// TIA Portal V18 export
FUNCTION "mot_speed_by_target" : Void   // FC7, FBD
{ S7_Optimized_Access := 'TRUE' }
VERSION : 0.1
// stored: AutoNumber true, IsIECCheckEnabled false, SetENOAutomatically false, UDAEnableTagReadback false
   VAR_INPUT
      isMultiturn : Bool;
      MultiTurnGoesFwdOnly : Bool;
      SET_SPD_ABS : Real;
      POS : Real;
      TARGET : Real;
      par_lim_fwd : Real;
      par_lim_rev : Real;
      par_speed_absmax : Real;
      par_dist_absmax : Real;
      par_speed_crawl : Real;
      par_dist_crawl : Real;
      par_dist_stop : Real;
   END_VAR
   VAR_OUTPUT
      speed_dir : Real;
      ER : Bool;
      ER_W : WString;
   END_VAR
   VAR_TEMP
      target_plus_TURN : Real;
      target_minus_TURN : Real;
      target_local : Real;
      dir_fwd : Bool;
      dir_rev : Bool;
      speed_fwd : Real;
      speed_rev : Real;
      set_spd_w_dir : Real;
      turn : Real;
      dist_to_target : Real;
      dist_to_target_plus_turn : Real;
      dist_to_target_minus_turn : Real;
      distance1 : Real;
      distance2plus : Real;
      turn_inv : Real;
      distance3minus : Real;
      closest0 : Bool;
      closest1Plus : Bool;
      closest2Minus : Bool;
      target_normal : Real;
   END_VAR
BEGIN

REGION Network 2 (SCL)
   IF "ER_0_root".ACK THEN
       #ER_W := WSTRING#'';
       #ER := false;

   END_IF;
   #turn := #par_lim_fwd - #par_lim_rev;
   #turn_inv := - #turn;
END_REGION

REGION Network 3
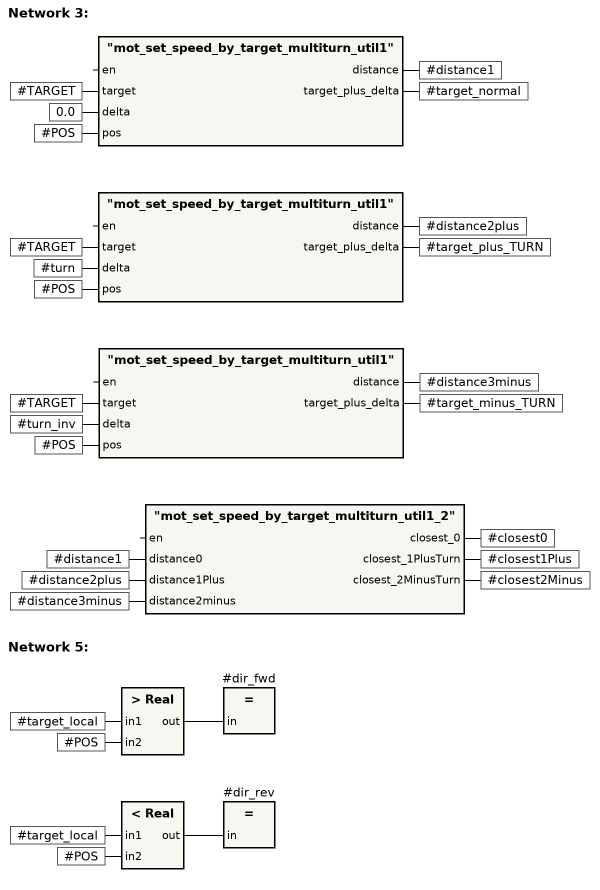
   "mot_set_speed_by_target_multiturn_util1"(target := #TARGET,
                           delta := 0.0,
                           pos := #POS,
                           distance => #distance1,
                           target_plus_delta => #target_normal);
   "mot_set_speed_by_target_multiturn_util1"(target := #TARGET,
                           delta := #turn,
                           pos := #POS,
                           distance => #distance2plus,
                           target_plus_delta => #target_plus_TURN);
   "mot_set_speed_by_target_multiturn_util1"(target := #TARGET,
                           delta := #turn_inv,
                           pos := #POS,
                           distance => #distance3minus,
                           target_plus_delta => #target_minus_TURN);
   "mot_set_speed_by_target_multiturn_util1_2"(distance0 := #distance1,
                           distance1Plus := #distance2plus,
                           distance2minus := #distance3minus,
                           closest_0 => #closest0,
                           closest_1PlusTurn => #closest1Plus,
                           closest_2MinusTurn => #closest2Minus);
END_REGION

REGION Network 4 (SCL)
   IF #isMultiturn AND NOT #ER THEN
       IF #MultiTurnGoesFwdOnly THEN
           IF #closest1Plus THEN
               #target_local := #target_plus_TURN;
           ELSE
               #target_local := #target_normal;
           END_IF;
       ELSE
           IF #closest1Plus THEN
               #target_local := #target_plus_TURN;
           ELSIF #closest2Minus THEN
               #target_local := #target_minus_TURN;
           ELSE
               #target_local := #target_normal;
           END_IF;
       END_IF;


   ELSE
       #target_local := #TARGET;
   END_IF;
END_REGION

REGION Network 5
   #dir_fwd := #target_local > #POS;
   #dir_rev := #target_local < #POS;
END_REGION

REGION Network 6
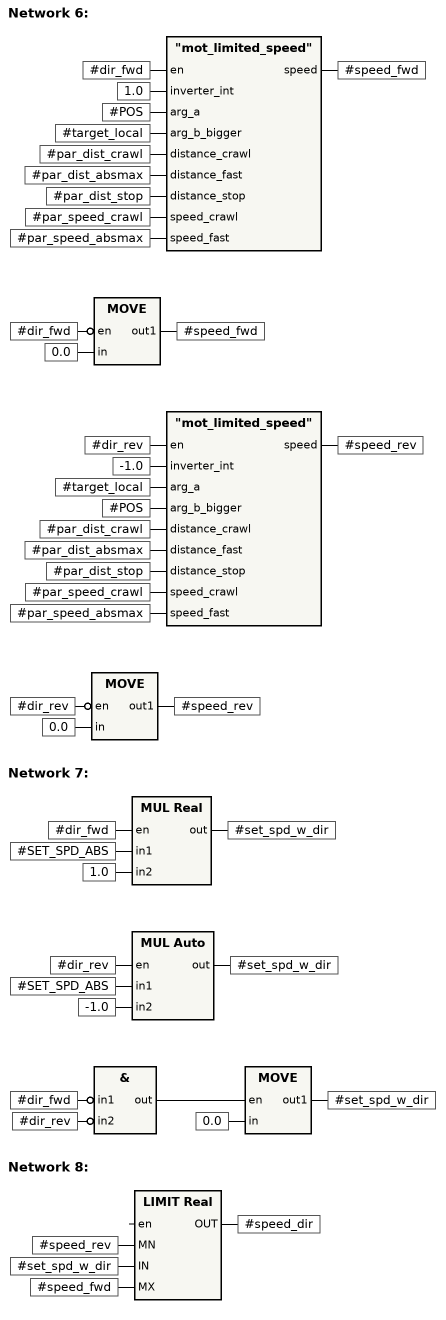
   IF #dir_fwd THEN
       "mot_limited_speed"(inverter_int := 1.0,
                           arg_a := #POS,
                           arg_b_bigger := #target_local,
                           distance_crawl := #par_dist_crawl,
                           distance_fast := #par_dist_absmax,
                           distance_stop := #par_dist_stop,
                           speed_crawl := #par_speed_crawl,
                           speed_fast := #par_speed_absmax,
                           speed => #speed_fwd);
   END_IF;
   IF NOT #dir_fwd THEN #speed_fwd := 0.0; END_IF;
   IF #dir_rev THEN
       "mot_limited_speed"(inverter_int := -1.0,
                           arg_a := #target_local,
                           arg_b_bigger := #POS,
                           distance_crawl := #par_dist_crawl,
                           distance_fast := #par_dist_absmax,
                           distance_stop := #par_dist_stop,
                           speed_crawl := #par_speed_crawl,
                           speed_fast := #par_speed_absmax,
                           speed => #speed_rev);
   END_IF;
   IF NOT #dir_rev THEN #speed_rev := 0.0; END_IF;
END_REGION

REGION Network 7
   IF #dir_fwd THEN #set_spd_w_dir := #SET_SPD_ABS * 1.0; END_IF;
   IF #dir_rev THEN #set_spd_w_dir := #SET_SPD_ABS * (-1.0); END_IF;
   IF NOT #dir_fwd AND NOT #dir_rev THEN #set_spd_w_dir := 0.0; END_IF;
END_REGION

REGION Network 8
   #speed_dir := LIMIT(MN := #speed_rev, IN := #set_spd_w_dir, MX := #speed_fwd);
END_REGION
END_FUNCTION
